PROGRAM Mapping_IO
VAR
END_VAR



G_IO.I_StartPushButton 				:= DeviceMapping.Input00_00;
G_IO.I_ResetPushButton 				:= DeviceMapping.Input00_01;
G_IO.I_StopPushButton 				:= DeviceMapping.Input00_02;






DeviceMapping.Output00_00 := G_IO.O_StartPushButton;
DeviceMapping.Output00_01 := G_IO.O_ResetPushButton;
DeviceMapping.Output00_02 := G_IO.O_StopPushButton;

END_PROGRAM

(* stored: Version 1.1.0.1, ProductVersion 3.1.4024.11
   POU Mapping_IO: Id {59b03e35-a5ac-47fe-bb36-b0cb5101e777}, SpecialFunc None *)
